(* CODESYS project sensata_data.library
   Company: Sensata Technologies
   Version: 1.0.1
   DocFormat: reStructuredText
   Placeholder: Sensata_Data
   Title: Sensata_Data

Project tree, tasks and I/O mapping:
  libraries: Sensata_Common, * (Sensata Technologies); Sensata_Utilities, * (Sensata Technologies); Tc2_Standard, * (Beckhoff Automation GmbH); Tc2_System, * (Beckhoff Automation GmbH); Tc2_Utilities, * (Beckhoff Automation GmbH); Tc3_JsonXml, * (Beckhoff Automation GmbH); Tc3_Module, * (Beckhoff Automation GmbH)
  Abstract/
    function block FB_Data [ST]: M_TransferData
    function block FB_MESData [ST]
  Concrete/
    data type E_DataTracker_Error
    function block FB_DataTracker [ST]: A_CommandRecovery, M_RouterHelper, M_TransferData
    function block FB_MESDataTracking [ST]: M_AddContactBlockQuantity, M_AddMachineResult, M_AddMachineWorkLoadTime, M_AddNewOperator, M_AddOutputTare, M_AddScrap, M_AddScrapComponentByReason, M_CheckContactBlock, M_CheckIncomingTare, M_ComponentsValidation, M_DTCTrayAddInfo, M_DTCTrayEmpty, M_DTCTrayGetInfo, M_EndLotComponent, M_EndLotOK, M_GetComponentInfoFromComponentBarCode, M_GetDrawingLink, M_GetInstructionLink, M_GetLotInfoFromLotBarCode, M_GetMachineDefects, M_GetMachineSettings, M_GetOperationLeftQty, M_GetOperatorInfoFromOperatorBarCode, M_GetProdLotComponents, M_GetRFIDAccess, M_StartLot, A_CommandRecovery, M_RouterHelper, M_TransferData
  MES_Structs/
    data type ComponentInfo
    data type ConnectionStringInfo
    data type DtcTrayInfo
    data type LotInfo
    data type OperationResult
    data type OperationResult_LotInfo
    data type ProductInfo
    data type ScrapInfo
    data type UserInfo
  Project Information/
    function F_GetCompany [ST]
    function F_GetTitle [ST]
    function F_GetVersion [ST]
  Version/
    global variables Global_Version
*)

// Concrete/E_DataTracker_Error
{attribute 'qualified_only'}
{attribute 'strict'}
TYPE E_DataTracker_Error :
(
	NoError := 0,
	DataStoringError :=100,
	DataReadingError := 101
) UDINT;
END_TYPE

// MES_Structs/ComponentInfo
TYPE ComponentInfo :
STRUCT
	ident        : LINT;    // Equivalent to C# long
    ident2       : DINT;    // Equivalent to C# int
    seria        : STRING;  // Equivalent to C# string
    quan         : DINT;    // Equivalent to C# int
    result       : INT;     // Equivalent to C# short
    resultText   : STRING;  // Equivalent to C# string
    actualQuan   : DINT;    // Equivalent to C# int
    item         : STRING;  // Equivalent to C# string
END_STRUCT
END_TYPE

// MES_Structs/ConnectionStringInfo
TYPE ConnectionStringInfo :
STRUCT
    UserID               : STRING;  // UserId for DB
    Password             : STRING;  // Password for user
    TraceabilityServer   : STRING;  // DB Server of Traceability
    TraceabilityDBName   : STRING;  // Database Name to use
    ApplicationName      : STRING;  // Name of application using TraceAbility
END_STRUCT
END_TYPE

// MES_Structs/DtcTrayInfo
TYPE DtcTrayInfo :
STRUCT
	Lot           : STRING;  // Production lot number
    Product       : STRING;  // Production lot item number
    Order         : STRING;  // Production lot order/job number. Type int on older version
    SNumber       : INT;     // Production seq number of lot in tray
    TrayStatus    : DINT;    // Production tray status - fail code or pass(0) or empty(-2)
    LastOperation : STRING;  // Last worked Operation
END_STRUCT
END_TYPE

// MES_Structs/LotInfo
(*
    Type: ST_LotInfo
    Support properties for lot information
*)
TYPE LotInfo :
STRUCT
	Lot           : STRING;  // Production lot number
    Product       : STRING;  // Production lot item number
    Order         : STRING;  // Production lot order/job number. Type int on older version
    Quantity      : DINT;    // Production lot qty
    Operator      : STRING;  // Operator ID from operator badge, working on lot
    ShiftLeader   : STRING;  // Static H param
    MachineID     : STRING;  // MachineID for TraceAbility
    LotIdent      : LINT;    // LotID for TraceAbility
    PiecesLeft    : DINT;    // LotID pcs left for work on machine
    PiecesOK      : DINT;    // Lot good pcs
    PiecesNOK     : DINT;    // Lot scrap pcs
END_STRUCT
END_TYPE

// MES_Structs/OperationResult
(*
    Type: T_OperationResult
    Support traceability results
*)
TYPE OperationResult :
STRUCT
    Success     : BOOL;        // Return if validation is passed successfully
    ErrorCode   : DINT;        // If there is error return code of error
    MessagesList: ARRAY [1..100] OF STRING;  // Return list of error messages if validation is not passed
    MsgCount    : DINT;        // Counter to keep track of the next empty slot in MessagesList
END_STRUCT
END_TYPE

// MES_Structs/OperationResult_LotInfo
TYPE OperationResult_LotInfo EXTENDS OperationResult :
STRUCT
//   Base         : OperationResult;  // Base OperationResult structure
//   ResultObject : LotInfo;           // Result object of type T_LotInfo
	test1 : OperationResult;
	ResultObject : LotInfo;
END_STRUCT
END_TYPE

// MES_Structs/ProductInfo
(*
    Type: T_ProductInfo
    Support properties for product information
*)
TYPE ProductInfo :
STRUCT
    ProductSetting   : STRING;  // Machine product values, + separator
    ProductStructure : STRING;  // Machine product structures, + separator
END_STRUCT
END_TYPE

// MES_Structs/ScrapInfo
(*
    Type: T_ScrapInfo
    Support properties for scrap information
*)
TYPE ScrapInfo :
STRUCT
    ScrapCode      : DINT;    // Scrap code number
    ScrapCount     : DINT;    // Scrap qty
    ScrapCodeDescr : STRING;  // Scrap code description
END_STRUCT
END_TYPE

// MES_Structs/UserInfo
(*
    Type: T_UserInfo
    Support properties for user information
*)
TYPE UserInfo :
STRUCT
    UserName    : STRING;  // User name
    AccessLevel : INT;     // Access Level
    UserID      : STRING;  // User name ID
    CardHash    : STRING;  // User card hash
END_STRUCT
END_TYPE

// Version/Global_Version
{attribute 'TcGenerated'}
{attribute 'no-analysis'}
{attribute 'linkalways'}
// This function has been automatically generated from the project information.
VAR_GLOBAL CONSTANT
	{attribute 'const_non_replaced'}
	stLibVersion_Sensata_Data : ST_LibVersion := (iMajor := 1, iMinor := 0, iBuild := 1, iRevision := 0, nFlags := 0, sVersion := '1.0.1');
END_VAR

// Abstract/FB_Data
FUNCTION_BLOCK ABSTRACT FB_Data EXTENDS FB_Module
VAR_INPUT
END_VAR
VAR_OUTPUT
END_VAR
VAR
END_VAR

METHOD M_TransferData : BOOL
(* starts the data transfer process for the provided dataPackege ID*)
VAR_INPUT
	(* Name of the data defineitoin *)
	_in_strDataPackageName : T_MaxString;
END_VAR
THIS^.M_LogWarning('M_TransferData not implemented!');
M_TransferData := TRUE;
END_METHOD

END_FUNCTION_BLOCK

// Abstract/FB_MESData
FUNCTION_BLOCK ABSTRACT FB_MESData EXTENDS FB_Module
VAR_INPUT
END_VAR
VAR_OUTPUT
END_VAR
VAR
END_VAR

END_FUNCTION_BLOCK

// Concrete/FB_DataTracker
(*
	Function block for reading and writing data from and to a persitatnt datastore.
	The mechanisms for data storage and retreiva are defined in the APT DataTracker mdules.
		
	First release: 2022-09-28 George Paiva <gpaiva@sensata.com>
*)
FUNCTION_BLOCK FB_DataTracker EXTENDS FB_Data
VAR_INPUT
	(* Reference to an FB_CommandRouter function block to send commands
	 	to a command router in the API. *)
	in_fbApi : REFERENCE TO FB_CommandRouter;
END_VAR
VAR_IN_OUT
END_VAR
VAR_OUTPUT
END_VAR
VAR CONSTANT
END_VAR
VAR
	bRouterBusy: BOOL; // TRUE while M_RouterHelper is being used by a method
	intRouterHelperStep: INT;
	intTransferDataStep: INT;
	bRouterHelperBusy: BOOL;
	bTransferDataBusy: BOOL;
END_VAR

A_CommandRecovery();

ACTION A_CommandRecovery:
IF NOT bRouterHelperBusy AND intRouterHelperStep > 0 THEN
	intRouterHelperStep := 0;
	THIS^.M_LogWarning('Router helper stopped prematurely!');
END_IF
bRouterHelperBusy := FALSE;

IF NOT bTransferDataBusy AND intTransferDataStep > 0 THEN
	intTransferDataStep := 0;
	bRouterBusy := FALSE;
	THIS^.M_LogWarning('Transfer data stopped prematurely!');
END_IF
bTransferDataBusy := FALSE;
END_ACTION

(*
Sends the given method to the API and receives and partially parses the result.
*)
METHOD PRIVATE M_RouterHelper : BOOL
VAR_INPUT
	(* Name of the method to call. *)
	_in_strMethodName : T_MaxString;
	(* Maximum time to wait for method response. *)
	_in_timeTimeout : TIME;
END_VAR
VAR_IN_OUT
	(* The array of parameters to send to the API. *)
	_inout_arrParams : T_ApiParameterList;
	(* The array that gets populated with any method output data. *)
	_inout_arrOutputs : T_ApiParameterList;
END_VAR
VAR_OUTPUT
	(* JSON string of the method return value. *)
	_out_strReturnValue: T_ApiParamValue;
END_VAR
VAR_INST
	(* Current step. *)
	_inst_intStep: INT;
	(* True if the method executed. *)
	_inst_bExec: BOOL;
	(* Return string of the method. *)
	_inst_strRet: T_ApiParamValue;
END_VAR
VAR
	(* True once the command routing finishes. *)
	_bComplete: BOOL;
	(* True once the API connects. *)
	_bApiConnect: BOOL;
END_VAR
_inst_intStep := intRouterHelperStep;
bRouterHelperBusy := TRUE;

CASE _inst_intStep OF
	0: // Start process only if there is no error on this FB
		IF NOT THIS^.P_bError THEN
			in_fbApi.M_ClearError();
			_inst_intStep := 10;
		END_IF
		
	10: // Check if command router connected
		IF NOT in_fbApi.P_bConnected THEN
			_inst_intStep := 20; // Go to API connect step
		ELSE
			_inst_intStep := 30; // Go to route command step
		END_IF
		
	20: // Connect the command router
		_bApiConnect := in_fbApi.M_Connect();
		IF _bApiConnect THEN
			_inst_intStep := _inst_intStep + 10; // Go to next step
		ELSIF in_fbApi.P_bError THEN
			THIS^.M_SetError(0, 'Error on command router function block while connecting!');
			_inst_intStep := 0; // Go back to start
		END_IF
		
	30:	// Route the command
		_bComplete := in_fbApi.M_RouteCommand(
			_in_strModuleId := in_strUniqueId,
			_in_strMethodName := _in_strMethodName,
			_in_timeTimeout := _in_timeTimeout,
			_inout_arrParameters := _inout_arrParams,
			_inout_arrOutputs := _inout_arrOutputs,
			_out_bCommandExecuted => _inst_bExec,
			_out_strReturnValue => _inst_strRet);
		IF _bComplete THEN
			_inst_intStep := _inst_intStep + 10; // Go to next step
		ELSIF in_fbApi.P_bError THEN
			THIS^.M_SetError(0, 'Error on command router function block while routing command!');
			_inst_intStep := 0; // Go back to start
		END_IF
		
	40: // Check result then go back to start
		IF NOT _inst_bExec THEN
			THIS^.M_SetError(0, 'Method in API failed to execute!');
		ELSE
			_out_strReturnValue := _inst_strRet;
			M_RouterHelper := TRUE;
		END_IF
		_inst_intStep := 0; // Go back to start
END_CASE
intRouterHelperStep := _inst_intStep;
END_METHOD

METHOD M_TransferData : BOOL
(* starts the data transfer process for the provided dataPackege ID*)
VAR_INPUT
	(* Name of the data defineitoin *)
	_in_strDataPackageName : T_MaxString;
END_VAR
VAR CONSTANT
	_strCOMMAND_NAME : T_MaxString	:= 'TransferData'; // Name of the API method
	_timeCOMMAND_TIMEOUT : TIME		:= T#30S; // Max time to receive API response
	_strSTART_MSG : T_MaxString		:= 'Retrieving Data'; // Prints when method starts
	_strEND_MSG : T_MaxString		:= 'Data Retrieval Complete'; // Prints when method finishes
	_udintERROR_ID : UDINT			:= E_DataTracker_Error.DataReadingError; // Error ID to set if command fails
	_strERROR_MSG : T_MaxString		:= 'Failed to store data!'; // Error message to set if command fails
END_VAR
VAR_INST
	_inst_arrParams: T_ApiParameterList; // Parameters array
	_inst_arrOutputs: T_ApiParameterList; // Outputs array
	_inst_strRet: T_ApiParamValue; // Return string from the router
	_inst_intStep: INT; // Current method step
	_inst_fbParams: FB_ApiParamBuilder; // Parameter builder FB
END_VAR
VAR
	_bComplete: BOOL; // True if the routing finishes
	_bResult : BOOL; // Output of the method
	_bRet: BOOL; //Return the bool value of the method
END_VAR
_inst_intStep := intTransferDataStep;
bTransferDataBusy := TRUE;

_bResult := FALSE;
CASE _inst_intStep OF
	0: // Wait for no error and router not busy
		IF NOT THIS^.P_bError AND NOT bRouterBusy THEN
			bRouterBusy := TRUE;
			_inst_intStep := _inst_intStep + 10;
		END_IF
		
	10: // Initialize parameters
		THIS^.M_LogMessage(_strSTART_MSG);
		_inst_fbParams.M_ClearParameters();
		// ADD ANY PARAMETERS HERE
		_inst_fbParams.M_AddParameter('itemName', _in_strDataPackageName);
		_inst_fbParams.M_OutputToParameterList(_inst_arrParams);
		_inst_intStep := _inst_intStep + 10;
		
	20: // Route the command
		_bComplete := M_RouterHelper(
			_in_strMethodName := _strCOMMAND_NAME, 
			_in_timeTimeout := _timeCOMMAND_TIMEOUT,
			_inout_arrParams := _inst_arrParams,
			_inout_arrOutputs := _inst_arrOutputs,
			_out_strReturnValue=>_inst_strRet);
		
		// If route completed, move to next step
		IF _bComplete THEN
			_inst_intStep := _inst_intStep + 10;
			bRouterBusy := FALSE;
		ELSIF THIS^.P_bError THEN
			_inst_intStep := 0;
			bRouterBusy := FALSE;
		END_IF
		
	30: // Parse results
		_bRet := STRING_TO_BOOL(_inst_strRet);		
		IF _bRet THEN
			_bResult := TRUE;
			THIS^.M_LogMessage(_strEND_MSG);
		// Set error if command failed
		ELSE
			THIS^.M_SetError(_udintERROR_ID, _strERROR_MSG);
		END_IF
		
		// Go back to start
		_inst_intStep := 0;
END_CASE
M_TransferData := _bResult;
intTransferDataStep := _inst_intStep;
END_METHOD

END_FUNCTION_BLOCK

// Concrete/FB_MESDataTracking
(*
	This function Block facilitates all the functinalities related to 
	MES Data Tracking Library on Sensata_Data C# API Library.
*)
FUNCTION_BLOCK FB_MESDataTracking EXTENDS FB_MESData
VAR_INPUT
	(* Reference to an FB_CommandRouter function block to send commands
	to a command router in the API. *)
	in_fbApi : REFERENCE TO FB_CommandRouter;
END_VAR
VAR_OUTPUT
END_VAR
VAR_IN_OUT
END_VAR
VAR_OUTPUT
END_VAR
VAR CONSTANT
END_VAR
VAR
	bRouterBusy: BOOL; // TRUE while M_RouterHelper is being used by a method
	intRouterHelperStep: INT;
	intGetLotInfoFromLotBarCodeStep: INT;
	bRouterHelperBusy: BOOL;
	intTransferDataStep: INT;
	bGetLotInfoFromLotBarCodeBusy: BOOL;
	bTransferDataBusy: BOOL;
END_VAR

A_CommandRecovery();

METHOD M_AddContactBlockQuantity : OperationResult
VAR_INPUT
END_VAR
END_METHOD

METHOD M_AddMachineResult : OperationResult
VAR_INPUT
END_VAR
END_METHOD

METHOD M_AddMachineWorkLoadTime : OperationResult
VAR_INPUT
END_VAR
END_METHOD

METHOD M_AddNewOperator : OperationResult
VAR_INPUT
END_VAR
END_METHOD

METHOD M_AddOutputTare : OperationResult
VAR_INPUT
END_VAR
END_METHOD

METHOD M_AddScrap : OperationResult
VAR_INPUT
END_VAR
END_METHOD

METHOD M_AddScrapComponentByReason : OperationResult
VAR_INPUT
END_VAR
END_METHOD

METHOD M_CheckContactBlock : OperationResult
VAR_INPUT
END_VAR
END_METHOD

METHOD M_CheckIncomingTare : OperationResult
VAR_INPUT
END_VAR
END_METHOD

METHOD M_ComponentsValidation : OperationResult
VAR_INPUT
END_VAR
END_METHOD

METHOD M_DTCTrayAddInfo : OperationResult
VAR_INPUT
END_VAR
END_METHOD

METHOD M_DTCTrayEmpty : OperationResult
VAR_INPUT
END_VAR
END_METHOD

METHOD M_DTCTrayGetInfo : OperationResult
VAR_INPUT
END_VAR
END_METHOD

METHOD M_EndLotComponent : OperationResult
VAR_INPUT
END_VAR
END_METHOD

METHOD M_EndLotOK : OperationResult
VAR_INPUT
END_VAR
END_METHOD

METHOD M_GetComponentInfoFromComponentBarCode : OperationResult
VAR_INPUT
END_VAR
END_METHOD

METHOD M_GetDrawingLink : OperationResult
VAR_INPUT
END_VAR
END_METHOD

METHOD M_GetInstructionLink : OperationResult
VAR_INPUT
END_VAR
END_METHOD

METHOD M_GetLotInfoFromLotBarCode : BOOL
VAR_INPUT
	lotBarCode : STRING;
END_VAR
VAR CONSTANT
	_strCOMMAND_NAME : T_MaxString	:= 'GetLotInfoFromLotBarCode'; // Name of the API method
	_timeCOMMAND_TIMEOUT : TIME		:= T#30S; // Max time to receive API response
	_strSTART_MSG : T_MaxString		:= 'Retrieving Data'; // Prints when method starts
	_strEND_MSG : T_MaxString		:= 'Data Retrieval Complete'; // Prints when method finishes
	_udintERROR_ID : UDINT			:= E_DataTracker_Error.DataReadingError; // Error ID to set if command fails
	_strERROR_MSG : T_MaxString		:= 'Failed to store data!'; // Error message to set if command fails
END_VAR
VAR_OUTPUT
//	result : OperationResult_LotInfo;
END_VAR
VAR
	_bComplete: BOOL; // True if the routing finishes
	_bResult : BOOL; // Output of the method
	_bRet: BOOL; //Return the bool value of the method
END_VAR
VAR_INST
	_inst_arrParams: T_ApiParameterList; // Parameters array
	_inst_arrOutputs: T_ApiParameterList; // Outputs array
	_inst_strRet: T_ApiParamValue; // Return string from the router
	_inst_intStep: INT; // Current method step
	_inst_fbParams: FB_ApiParamBuilder; // Parameter builder FB
END_VAR
_inst_intStep := intGetLotInfoFromLotBarCodeStep;
bGetLotInfoFromLotBarCodeBusy := TRUE;

_bResult := FALSE;
CASE _inst_intStep OF
	0: // Wait for no error and router not busy
		IF NOT THIS^.P_bError AND NOT bRouterBusy THEN
			bRouterBusy := TRUE;
			_inst_intStep := _inst_intStep + 10;
		END_IF
		
	10: // Initialize parameters
		THIS^.M_LogMessage(_strSTART_MSG);
		_inst_fbParams.M_ClearParameters();
		// ADD ANY PARAMETERS HERE
		_inst_fbParams.M_AddParameter('lotBarCode', lotBarCode);
		_inst_fbParams.M_OutputToParameterList(_inst_arrParams);
		_inst_intStep := _inst_intStep + 10;
		
	20: // Route the command
		_bComplete := M_RouterHelper(
			_in_strMethodName := _strCOMMAND_NAME, 
			_in_timeTimeout := _timeCOMMAND_TIMEOUT,
			_inout_arrParams := _inst_arrParams,
			_inout_arrOutputs := _inst_arrOutputs,
			_out_strReturnValue=>_inst_strRet);
		
		// If route completed, move to next step
		IF _bComplete THEN
			_inst_intStep := _inst_intStep + 10;
			bRouterBusy := FALSE;
		ELSIF THIS^.P_bError THEN
			_inst_intStep := 0;
			bRouterBusy := FALSE;
		END_IF
		
	30: // Parse results
		_bRet := STRING_TO_BOOL(_inst_strRet);		
		IF _bRet THEN
			_bResult := TRUE;
			THIS^.M_LogMessage(_strEND_MSG);
		// Set error if command failed
		ELSE
			THIS^.M_SetError(_udintERROR_ID, _strERROR_MSG);
		END_IF
		
		// Go back to start
		_inst_intStep := 0;
END_CASE
M_GetLotInfoFromLotBarCode := _bResult;
intGetLotInfoFromLotBarCodeStep := _inst_intStep;
END_METHOD

METHOD M_GetMachineDefects : OperationResult
VAR_INPUT
END_VAR
END_METHOD

METHOD M_GetMachineSettings : OperationResult
VAR_INPUT
END_VAR
END_METHOD

METHOD M_GetOperationLeftQty : OperationResult
VAR_INPUT
END_VAR
END_METHOD

METHOD M_GetOperatorInfoFromOperatorBarCode : OperationResult
VAR_INPUT
END_VAR
END_METHOD

METHOD M_GetProdLotComponents : OperationResult
VAR_INPUT
END_VAR
END_METHOD

METHOD M_GetRFIDAccess : OperationResult
VAR_INPUT
END_VAR
END_METHOD

METHOD M_StartLot : OperationResult
VAR_INPUT
END_VAR
END_METHOD

ACTION A_CommandRecovery:
IF NOT bRouterHelperBusy AND intRouterHelperStep > 0 THEN
	intRouterHelperStep := 0;
	THIS^.M_LogWarning('Router helper stopped prematurely!');
END_IF
bRouterHelperBusy := FALSE;

IF NOT bTransferDataBusy AND intTransferDataStep > 0 THEN
	intTransferDataStep := 0;
	bRouterBusy := FALSE;
	THIS^.M_LogWarning('Transfer data stopped prematurely!');
END_IF
bTransferDataBusy := FALSE;
END_ACTION

(*
Sends the given method to the API and receives and partially parses the result.
*)
METHOD PRIVATE M_RouterHelper : BOOL
VAR_INPUT
	(* Name of the method to call. *)
	_in_strMethodName : T_MaxString;
	(* Maximum time to wait for method response. *)
	_in_timeTimeout : TIME;
END_VAR
VAR_IN_OUT
	(* The array of parameters to send to the API. *)
	_inout_arrParams : T_ApiParameterList;
	(* The array that gets populated with any method output data. *)
	_inout_arrOutputs : T_ApiParameterList;
END_VAR
VAR_OUTPUT
	(* JSON string of the method return value. *)
	_out_strReturnValue: T_ApiParamValue;
END_VAR
VAR_INST
	(* Current step. *)
	_inst_intStep: INT;
	(* True if the method executed. *)
	_inst_bExec: BOOL;
	(* Return string of the method. *)
	_inst_strRet: T_ApiParamValue;
END_VAR
VAR
	(* True once the command routing finishes. *)
	_bComplete: BOOL;
	(* True once the API connects. *)
	_bApiConnect: BOOL;
END_VAR
_inst_intStep := intRouterHelperStep;
bRouterHelperBusy := TRUE;

CASE _inst_intStep OF
	0: // Start process only if there is no error on this FB
		IF NOT THIS^.P_bError THEN
			in_fbApi.M_ClearError();
			_inst_intStep := 10;
		END_IF
		
	10: // Check if command router connected
		IF NOT in_fbApi.P_bConnected THEN
			_inst_intStep := 20; // Go to API connect step
		ELSE
			_inst_intStep := 30; // Go to route command step
		END_IF
		
	20: // Connect the command router
		_bApiConnect := in_fbApi.M_Connect();
		IF _bApiConnect THEN
			_inst_intStep := _inst_intStep + 10; // Go to next step
		ELSIF in_fbApi.P_bError THEN
			THIS^.M_SetError(0, 'Error on command router function block while connecting!');
			_inst_intStep := 0; // Go back to start
		END_IF
		
	30:	// Route the command
		_bComplete := in_fbApi.M_RouteCommand(
			_in_strModuleId := in_strUniqueId,
			_in_strMethodName := _in_strMethodName,
			_in_timeTimeout := _in_timeTimeout,
			_inout_arrParameters := _inout_arrParams,
			_inout_arrOutputs := _inout_arrOutputs,
			_out_bCommandExecuted => _inst_bExec,
			_out_strReturnValue => _inst_strRet);
		IF _bComplete THEN
			_inst_intStep := _inst_intStep + 10; // Go to next step
		ELSIF in_fbApi.P_bError THEN
			THIS^.M_SetError(0, 'Error on command router function block while routing command!');
			_inst_intStep := 0; // Go back to start
		END_IF
		
	40: // Check result then go back to start
		IF NOT _inst_bExec THEN
			THIS^.M_SetError(0, 'Method in API failed to execute!');
		ELSE
			_out_strReturnValue := _inst_strRet;
			M_RouterHelper := TRUE;
		END_IF
		_inst_intStep := 0; // Go back to start
END_CASE
intRouterHelperStep := _inst_intStep;
END_METHOD

METHOD M_TransferData : BOOL
(* starts the data transfer process for the provided dataPackege ID*)
VAR_INPUT
	(* Name of the data defineitoin *)
	_in_strDataPackageName : T_MaxString;
END_VAR
VAR CONSTANT
	_strCOMMAND_NAME : T_MaxString	:= 'TransferData'; // Name of the API method
	_timeCOMMAND_TIMEOUT : TIME		:= T#30S; // Max time to receive API response
	_strSTART_MSG : T_MaxString		:= 'Retrieving Data'; // Prints when method starts
	_strEND_MSG : T_MaxString		:= 'Data Retrieval Complete'; // Prints when method finishes
	_udintERROR_ID : UDINT			:= E_DataTracker_Error.DataReadingError; // Error ID to set if command fails
	_strERROR_MSG : T_MaxString		:= 'Failed to store data!'; // Error message to set if command fails
END_VAR
VAR_INST
	_inst_arrParams: T_ApiParameterList; // Parameters array
	_inst_arrOutputs: T_ApiParameterList; // Outputs array
	_inst_strRet: T_ApiParamValue; // Return string from the router
	_inst_intStep: INT; // Current method step
	_inst_fbParams: FB_ApiParamBuilder; // Parameter builder FB
END_VAR
VAR
	_bComplete: BOOL; // True if the routing finishes
	_bResult : BOOL; // Output of the method
	_bRet: BOOL; //Return the bool value of the method
	_pStructPointer : PVOID; // Pointer to the struct
	intIndex : INT;
END_VAR
VAR_OUTPUT
	_out_bSuccess : BOOL;
	_out_intErrorCode : DINT;
	_out_arrstrMessageList : ARRAY[0..10] OF T_MaxString;
END_VAR

_inst_intStep := intTransferDataStep;
bTransferDataBusy := TRUE;

_bResult := FALSE;
CASE _inst_intStep OF
	0: // Wait for no error and router not busy
		IF NOT THIS^.P_bError AND NOT bRouterBusy THEN
			bRouterBusy := TRUE;
			_inst_intStep := _inst_intStep + 10;
		END_IF
		
	10: // Initialize parameters
		THIS^.M_LogMessage(_strSTART_MSG);
		_inst_fbParams.M_ClearParameters();
		// ADD ANY PARAMETERS HERE
		_inst_fbParams.M_AddParameter('itemName', _in_strDataPackageName);
		_inst_fbParams.M_OutputToParameterList(_inst_arrParams);
		_inst_intStep := _inst_intStep + 10;
		
	20: // Route the command
		_bComplete := M_RouterHelper(
			_in_strMethodName := _strCOMMAND_NAME, 
			_in_timeTimeout := _timeCOMMAND_TIMEOUT,
			_inout_arrParams := _inst_arrParams,
			_inout_arrOutputs := _inst_arrOutputs,
			_out_strReturnValue=>_inst_strRet);
		
		// If route completed, move to next step
		IF _bComplete THEN
			_inst_intStep := _inst_intStep + 10;
			bRouterBusy := FALSE;
		ELSIF THIS^.P_bError THEN
			_inst_intStep := 0;
			bRouterBusy := FALSE;
		END_IF
		
	30: // Parse results
		_bRet := STRING_TO_BOOL(_inst_strRet);		
		IF _bRet THEN
			_bResult := TRUE;
			THIS^.M_LogMessage(_strEND_MSG);
			_inst_fbParams.M_LoadFromParameterList(_inst_arrOutputs);
			_out_bSuccess := _inst_fbParams.M_ParseBool(_inst_fbParams.M_GetParameter('_out_bSuccess'));
			_out_intErrorCode := _inst_fbParams.M_ParseInt(_inst_fbParams.M_GetParameter('_out_intErrorCode'));
			
		(* Get a pointer to an array parameter. Arrays cannot be fully parsed
			automatically, so each element of the array must be parsed individually. *)
		_pStructPointer := _inst_fbParams.M_GetStructMember(_pStructPointer, '_out_arrstrMessageList');
		
		(* Individual parse each array element *)
		FOR intIndex := 1 TO 10 DO
			_out_arrstrMessageList[intIndex] := _inst_fbParams.M_ParseString(_inst_fbParams.M_GetArrayElement(_pStructPointer, INT_TO_UDINT(intIndex)));
		END_FOR
			
		// Set error if command failed
		ELSE
			THIS^.M_SetError(_udintERROR_ID, _strERROR_MSG);
		END_IF
		
		// Go back to start
		_inst_intStep := 0;
END_CASE
M_TransferData := _bResult;
intTransferDataStep := _inst_intStep;
END_METHOD

END_FUNCTION_BLOCK

// Project Information/F_GetCompany
// This function has been automatically generated from the project information.
{attribute 'signature_flag' := '1073741824'}
{attribute 'TcGenerated'}
{attribute 'no-analysis'}
FUNCTION F_GetCompany : WSTRING
VAR_INPUT
	
END_VAR

F_GetCompany := "Sensata Technologies";

END_FUNCTION

// Project Information/F_GetTitle
// This function has been automatically generated from the project information.
{attribute 'signature_flag' := '1073741824'}
{attribute 'TcGenerated'}
{attribute 'no-analysis'}
FUNCTION F_GetTitle : WSTRING
VAR_INPUT
	
END_VAR

F_GetTitle := "Sensata_Data";

END_FUNCTION

// Project Information/F_GetVersion
// This function has been automatically generated from the project information.
{attribute 'signature_flag' := '1073741824'}
{attribute 'TcGenerated'}
{attribute 'no-analysis'}
FUNCTION F_GetVersion : ST_LibVersion
VAR_INPUT
	
END_VAR

F_GetVersion.iMajor := 1;
F_GetVersion.iMinor := 0;
F_GetVersion.iBuild := 1;
F_GetVersion.iRevision := 0;
F_GetVersion.sVersion := '1.0.1';
F_GetVersion.nFlags := 0;

END_FUNCTION
